	arCurrDataPoint.arFrequency_2:=arFrequency[2];
	arCurrDataPoint.arVoltage_L_N_2:=arVoltage_L_N[2];
	arCurrDataPoint.arCurrent_2:=arCurrent[2];
	arCurrDataPoint.arPower_2:=arCurrDataPoint.arCurrent_2*arCurrDataPoint.arVoltage_L_N_2;


	arCurrDataPoint.arFrequency_3:=arFrequency[3];
	arCurrDataPoint.arVoltage_L_N_3:=arVoltage_L_N[3];
	arCurrDataPoint.arCurrent_3:=arCurrent[3];
	arCurrDataPoint.arPower_3:=arCurrDataPoint.arCurrent_3*arCurrDataPoint.arVoltage_L_N_3;

	arCurrDataPoint.timeStamp := Get_Time();

	arCurrDataPoint.DCV1 := DCV1;
	arCurrDataPoint.DCV2:=DCV2;
	arCurrDataPoint.DCPower1:=DCPower1;
	arCurrDataPoint.DCPower2:=DCPower2;
	arCurrDataPoint.DCCurr2:=DCCurr2;
	arCurrDataPoint.DCCurr2:=DCCurr2;


	Create_Data_Point := arCurrDataPoint;
END_FUNCTION

(* POU 06. Mysql Write/Get_Time, ST *)
FUNCTION Get_Time : REAL
VAR_INPUT

END_VAR
VAR



END_VAR
(* Haal de systeemtijd op *)
Get_Time := DT_TO_REAL(SysRtcGetTime(FALSE));
END_FUNCTION

(* Visualisation power
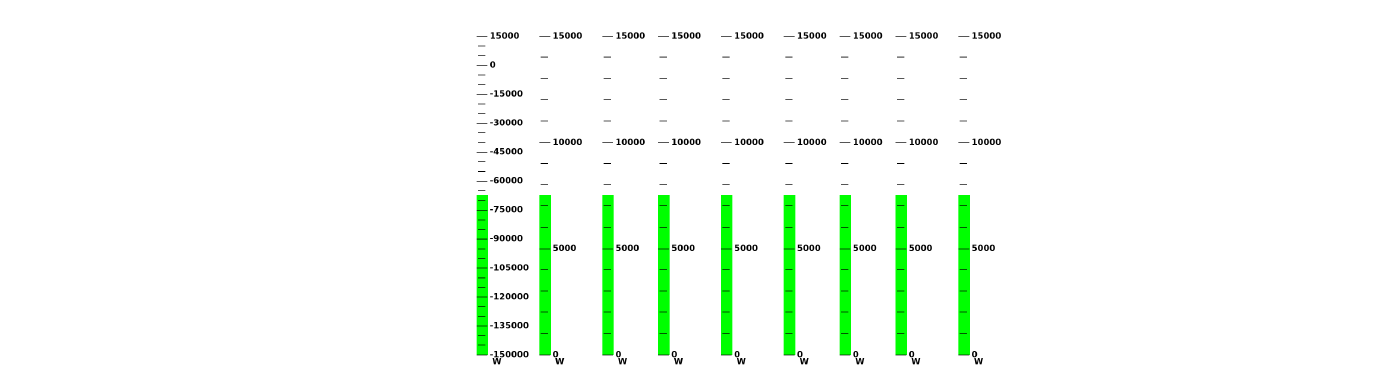
group at (20,60)-(91,571)
  rectangle at (0,0)-(1,1): text "{ExtendedElement},Visu\ElementDLL.ete,1,@Bargraph,71,511,1,1,0,PQ_1.rTotalActivePower,W,%.0f,5000,15000,-150000,15000,0,0,0,0,0,0,0,-13,16,700,Arial,0,255,0,255,0,0,0,0,0,0,0,0,0,,1,0,0,"
  rectangle at (11,248)-(26,463): alarm colour if (PQ_1.rTotalActivePower) < 0; top ((PQ_1.rTotalActivePower * 1.0) - -67500)  * -0.00260606
  rectangle at (27,452)-(66,473): text "-150000"
  rectangle at (27,413)-(66,434): text "-135000"
  rectangle at (27,374)-(66,395): text "-120000"
  rectangle at (27,335)-(66,356): text "-105000"
  rectangle at (27,296)-(66,317): text "-90000"
  rectangle at (27,257)-(66,278): text "-75000"
  rectangle at (27,218)-(66,239): text "-60000"
  rectangle at (27,179)-(66,200): text "-45000"
  rectangle at (27,140)-(66,161): text "-30000"
  rectangle at (27,101)-(66,122): text "-15000"
  rectangle at (27,62)-(66,83): text "0"
  rectangle at (27,23)-(66,44): text "15000"
  rectangle at (25,464)-(51,480): text "W"
group at (110,60)-(181,571)
  rectangle at (0,0)-(1,1): text "{ExtendedElement},Visu\ElementDLL.ete,1,@Bargraph,71,511,1,1,0,PQ_2.rTotalActivePower,W,%.0f,1000,5000,0,15000,0,0,0,0,0,0,0,-13,16,700,Arial,0,255,0,255,0,0,0,0,0,0,0,0,0,,1,0,0,"
  rectangle at (11,248)-(26,463): alarm colour if (PQ_2.rTotalActivePower) < 0; top ((PQ_2.rTotalActivePower * 1.0) - 7500)  * -0.0286667
  rectangle at (27,452)-(66,473): text "0"
  rectangle at (27,309)-(66,330): text "5000"
  rectangle at (27,166)-(66,187): text "10000"
  rectangle at (27,23)-(66,44): text "15000"
  rectangle at (25,464)-(51,480): text "W"
group at (200,60)-(271,571)
  rectangle at (0,0)-(1,1): text "{ExtendedElement},Visu\ElementDLL.ete,1,@Bargraph,71,511,1,1,0,PQ_3.rTotalActivePower,W,%.0f,1000,5000,0,15000,0,0,0,0,0,0,0,-13,16,700,Arial,0,255,0,255,0,0,0,0,0,0,0,0,0,,1,0,0,"
  rectangle at (11,248)-(26,463): alarm colour if (PQ_3.rTotalActivePower) < 0; top ((PQ_3.rTotalActivePower * 1.0) - 7500)  * -0.0286667
  rectangle at (27,452)-(66,473): text "0"
  rectangle at (27,309)-(66,330): text "5000"
  rectangle at (27,166)-(66,187): text "10000"
  rectangle at (27,23)-(66,44): text "15000"
  rectangle at (25,464)-(51,480): text "W"
group at (280,60)-(351,571)
  rectangle at (0,0)-(1,1): text "{ExtendedElement},Visu\ElementDLL.ete,1,@Bargraph,71,511,1,1,0,PQ_4.rTotalActivePower,W,%.0f,1000,5000,0,15000,0,0,0,0,0,0,0,-13,16,700,Arial,0,255,0,255,0,0,0,0,0,0,0,0,0,,1,0,0,"
  rectangle at (11,248)-(26,463): alarm colour if (PQ_4.rTotalActivePower) < 0; top ((PQ_4.rTotalActivePower * 1.0) - 7500)  * -0.0286667
  rectangle at (27,452)-(66,473): text "0"
  rectangle at (27,309)-(66,330): text "5000"
  rectangle at (27,166)-(66,187): text "10000"
  rectangle at (27,23)-(66,44): text "15000"
  rectangle at (25,464)-(51,480): text "W"
group at (370,60)-(441,571)
  rectangle at (0,0)-(1,1): text "{ExtendedElement},Visu\ElementDLL.ete,1,@Bargraph,71,511,1,1,0,PQ_5.rTotalActivePower,W,%.0f,1000,5000,0,15000,0,0,0,0,0,0,0,-13,16,700,Arial,0,255,0,255,0,0,0,0,0,0,0,0,0,,1,0,0,"
  rectangle at (11,248)-(26,463): alarm colour if (PQ_5.rTotalActivePower) < 0; top ((PQ_5.rTotalActivePower * 1.0) - 7500)  * -0.0286667
  rectangle at (27,452)-(66,473): text "0"
  rectangle at (27,309)-(66,330): text "5000"
  rectangle at (27,166)-(66,187): text "10000"
  rectangle at (27,23)-(66,44): text "15000"
  rectangle at (25,464)-(51,480): text "W"
group at (460,60)-(531,571)
  rectangle at (0,0)-(1,1): text "{ExtendedElement},Visu\ElementDLL.ete,1,@Bargraph,71,511,1,1,0,PQ_6.rTotalActivePower,W,%.0f,1000,5000,0,15000,0,0,0,0,0,0,0,-13,16,700,Arial,0,255,0,255,0,0,0,0,0,0,0,0,0,,1,0,0,"
  rectangle at (11,248)-(26,463): alarm colour if (PQ_6.rTotalActivePower) < 0; top ((PQ_6.rTotalActivePower * 1.0) - 7500)  * -0.0286667
  rectangle at (27,452)-(66,473): text "0"
  rectangle at (27,309)-(66,330): text "5000"
  rectangle at (27,166)-(66,187): text "10000"
  rectangle at (27,23)-(66,44): text "15000"
  rectangle at (25,464)-(51,480): text "W"
group at (540,60)-(611,571)
  rectangle at (0,0)-(1,1): text "{ExtendedElement},Visu\ElementDLL.ete,1,@Bargraph,71,511,1,1,0,PQ_7.rTotalActivePower,W,%.0f,1000,5000,0,15000,0,0,0,0,0,0,0,-13,16,700,Arial,0,255,0,255,0,0,0,0,0,0,0,0,0,,1,0,0,"
  rectangle at (11,248)-(26,463): alarm colour if (PQ_7.rTotalActivePower) < 0; top ((PQ_7.rTotalActivePower * 1.0) - 7500)  * -0.0286667
  rectangle at (27,452)-(66,473): text "0"
  rectangle at (27,309)-(66,330): text "5000"
  rectangle at (27,166)-(66,187): text "10000"
  rectangle at (27,23)-(66,44): text "15000"
  rectangle at (25,464)-(51,480): text "W"
group at (620,60)-(691,571)
  rectangle at (0,0)-(1,1): text "{ExtendedElement},Visu\ElementDLL.ete,1,@Bargraph,71,511,1,1,0,PQ_8.rTotalActivePower,W,%.0f,1000,5000,0,15000,0,0,0,0,0,0,0,-13,16,700,Arial,0,255,0,255,0,0,0,0,0,0,0,0,0,,1,0,0,"
  rectangle at (11,248)-(26,463): alarm colour if (PQ_8.rTotalActivePower) < 0; top ((PQ_8.rTotalActivePower * 1.0) - 7500)  * -0.0286667
  rectangle at (27,452)-(66,473): text "0"
  rectangle at (27,309)-(66,330): text "5000"
  rectangle at (27,166)-(66,187): text "10000"
  rectangle at (27,23)-(66,44): text "15000"
  rectangle at (25,464)-(51,480): text "W"
group at (710,60)-(781,571)
  rectangle at (0,0)-(1,1): text "{ExtendedElement},Visu\ElementDLL.ete,1,@Bargraph,71,511,1,1,0,PQ_9.rTotalActivePower,W,%.0f,1000,5000,0,15000,0,0,0,0,0,0,0,-13,16,700,Arial,0,255,0,255,0,0,0,0,0,0,0,0,0,,1,0,0,"
  rectangle at (11,248)-(26,463): alarm colour if (PQ_9.rTotalActivePower) < 0; top ((PQ_9.rTotalActivePower * 1.0) - 7500)  * -0.0286667
  rectangle at (27,452)-(66,473): text "0"
  rectangle at (27,309)-(66,330): text "5000"
  rectangle at (27,166)-(66,187): text "10000"
  rectangle at (27,23)-(66,44): text "15000"
  rectangle at (25,464)-(51,480): text "W"
162 more shapes without text or variables
*)
